// TwinCAT 3 PLC project SendingMQTT
// ProgramVersion: 3.1.4022.3
// libraries:
//   Tc2_Standard, * (Beckhoff Automation GmbH)
//   Tc2_System, * (Beckhoff Automation GmbH)
//   Tc2_Utilities, * (Beckhoff Automation GmbH)
//   Tc3_IotBase, * (Beckhoff Automation GmbH)
//   Tc3_IotCommunicator, * (Beckhoff Automation GmbH)
//   Tc3_JsonXml, * (Beckhoff Automation GmbH)
//   Tc3_Module, * (Beckhoff Automation GmbH)
// project tree:
//   DUTs/ HaDevice_1.TcDUT, HaProduct.TcDUT, TemperatureStructure.TcDUT, HaDevice.TcDUT
//   / PlcTask.TcTTO (not stored)
//   POUs/ MAIN.TcPOU
// real-time tasks:
//   TASK PlcTask: cycle T#10ms, priority 20, ADS port 350
// I/O:
//   DEVICE Device 2 (EtherCAT) (disabled), AmsNetId 192.168.250.2.3.1
//     Term 1 (EK1100) [EK1100 EtherCAT Coupler (2A E-Bus)]
//       Term 2 (EL1008) [EL1008 8Ch. Dig. Input 24V, 3ms]
//       Term 3 (EL2008) [EL2008 8Ch. Dig. Output 24V, 0.5A]
//       Term 4 (EL3314) [EL3314 4Ch. Ana. Input Thermocouple (TC)]
//       Term 5 (EL9011) [EL9011 End Terminal]
// variable links:
//   SendingMQTT/SendingMQTT Instance <-> Device 2 (EtherCAT)/Term 1 (EK1100)/Term 4 (EL3314)
//     PlcTask Inputs/MAIN.ai_RoomTemperature <-> TC Inputs Channel 1/Value

// ---- DUTs/HaDevice_1.TcDUT
TYPE HaDevice_1 :
STRUCT
	status		:	REAL;
	sensor1		:	REAL;
	sensor2		:	REAL;
	sensor12	:	REAL;
END_STRUCT
END_TYPE

// ---- DUTs/HaProduct.TcDUT
TYPE HaProduct :
STRUCT
	name			:	STRING;
	identifiers		:	ARRAY[1..1] OF STRING := ['smart dims'];
	model			:	STRING;
	manufacturer	:	STRING;
END_STRUCT
END_TYPE

// ---- DUTs/TemperatureStructure.TcDUT
TYPE TemperatureStructure :
STRUCT
	RoomTemperature : REAL;
	BathRoomTemperature : REAL;
	SomeOtherData : DINT;
	ekstra	: HaProduct;
END_STRUCT
END_TYPE

// ---- DUTs/HaDevice.TcDUT
TYPE HaDevice :
STRUCT
	name			:	STRING;
	state_topic		:	STRING;
	value_template	:	STRING;
	unique_id		:	STRING;
	device			: 	HaProduct;
END_STRUCT
END_TYPE

// ---- POUs/MAIN.TcPOU
PROGRAM MAIN
VAR
	fbMqttClient: FB_IotMqttClient; // MQTT client.       
    TopicToPublish   : STRING(255) := 'Temperatures'; // Mqtt topic on which we will broadcast the acual temperatures
    MessageToPublish : STRING(255); //String to send.
    fbSendMessageIntervalTimer : TON := (PT:=T#1S);	//Interval timer for broadcasting.
	ai_RoomTemperature AT %I* : INT; //Actual room temperature, linked to thermocouple	 
	
	TopicToPublishJson   : STRING(255) := 'unit1201/state'; //'homeassistant/sensor/unit_1400/config'; //'unit1201/state'; // Mqtt topic on which we will broadcast the acual temperatures in JSON format
	MessageToPublishJson : STRING(255); //String to send in JSON format
	mess				: STRING(1000) := '{"status":101}';
	//mess				: STRING ;
	fbJsonWriter : FB_JsonSaxWriter;
	fbJsonDataType : FB_JsonReadWriteDataType;
	TemperatureStructure:TemperatureStructure; 
	hadevice	:	HaDevice_1;	
	
	icount	:	INT;
	
	
	/// homeassistant/sensor/unit_1201/config
	
	(*
	{
  "name": "turned on",
  "state_topic": "unit1201/state",
  "unique_id": "unit_1201",
  "device": {
    "name": "smart enhed",
    "identifiers": [
      "unit_1201"
    ]
  }
}

"value_template": {% raw %}"{{ value_json.status }}"{% endraw %},
*)
	  


END_VAR

//mess := F_RTrim(mess1);

(*
hadevice.name			:= 'sensor2024';
hadevice.state_topic	:= 'unit1201/state';
hadevice.unique_id		:= 'unit_1400';
hadevice.value_template	:= '{{value_json.sensor2024 | round(2)}}';
hadevice.device.name	:= 'smart_enhed';
hadevice.device.identifiers[1]	:= 'smart_enhed';
hadevice.device.model			:= 'twincat3';
hadevice.device.manufacturer	:= 'beckhoff';
*)
IF _TaskInfo[GETCURTASKINDEXEX()].FirstCycle THEN    
    fbMqttClient.sHostName      := 'homeassistant'; // 192.168.2.159 - 100.97.177.128 - tailscale ip 100.92.234.119 - homeassistant
    fbMqttClient.nHostPort      := 1883;
	fbMqttClient.sUserName		:= 'twincat_xar';
	fbMqttClient.sUserPassword	:= '1234';
    fbMqttClient.sTopicPrefix   := '';     
	//fbMqttClient.sClientId 		:= 'Publishing PLC';
END_IF

fbMqttClient.Execute(TRUE);

IF fbMqttClient.bConnected THEN
    fbSendMessageIntervalTimer(IN:=TRUE);
    IF fbSendMessageIntervalTimer.Q THEN
        fbSendMessageIntervalTimer(IN:=FALSE);        
        MessageToPublish := CONCAT('Room temperature: ',REAL_TO_STRING(ai_RoomTemperature / 10.0));
		
        fbMqttClient.Publish(sTopic:= TopicToPublish, 
        	pPayload:= ADR(MessageToPublish), 
			nPayloadSize:= LEN2(ADR(MessageToPublish))+1, 
            eQoS:= TcIotMqttQos.AtMostOnceDelivery, 
			bRetain:= FALSE,
			bQueue:= FALSE);

			
			// Fill data
			IF hadevice.status <100 THEN
				hadevice.status := hadevice.status+1.11;
			END_IF
			IF hadevice.status > 20 THEN
			hadevice.status := 0;
			END_IF
			
			hadevice.sensor1 := 54;
			
			CASE icount OF
				0:
				IF hadevice.sensor2 <100 THEN
				hadevice.sensor2 := hadevice.sensor2+1;
				END_IF
				IF hadevice.sensor2 >= 20 THEN
					icount := 10;
				END_IF
				10:
				hadevice.sensor2 := hadevice.sensor2-1;
				IF hadevice.sensor2 <= 0 THEN
					icount := 0;
				END_IF
			END_CASE
			
		hadevice.sensor12 := 2024;	
	
			
			
			// COnvert to JSON string
			fbJsonWriter.ResetDocument();
			fbJsonDataType.AddJsonValueFromSymbol(fbJsonWriter, 'hadevice_1', SIZEOF(hadevice), ADR(hadevice));
			MessageToPublishJson := fbJsonWriter.GetDocument();
			fbJsonWriter.EndObject();
			fbJsonWriter.ResetDocument();
			
			//Publish
			fbMqttClient.Publish(sTopic:= TopicToPublishJson, 
        	pPayload:= ADR(MessageToPublishJson), 
			nPayloadSize:= LEN2(ADR(MessageToPublishJson)), 
            eQoS:= TcIotMqttQos.AtMostOnceDelivery, 
			bRetain:= FALSE,
			bQueue:= FALSE);
    END_IF
END_IF

TcIotMqttQos.AtLeastOnceDelivery;

END_PROGRAM
